FUNCTION_BLOCK StubXts EXTENDS Xts
VAR
END_VAR

METHOD Cycle : HRESULT
END_METHOD

METHOD Initialise : HRESULT
END_METHOD

METHOD MoverHomeSequence : BOOL
END_METHOD

METHOD SetDisabled : BOOL
VAR_INPUT
END_VAR
_XtsEnabled := FALSE;
END_METHOD

METHOD setEnabled : BOOL
VAR_INPUT
END_VAR
_XtsEnabled := TRUE;
END_METHOD

METHOD setInitialised : BOOL
VAR_INPUT
END_VAR
_Initialised := TRUE;
END_METHOD

METHOD setMoverNumberMax : BOOL
VAR_INPUT
END_VAR
_registeredNumberOfMovers := 255;
END_METHOD

METHOD setMoverNumberZero : BOOL
VAR_INPUT
END_VAR
_registeredNumberOfMovers := 0;
END_METHOD

METHOD setNotInitialised : BOOL
VAR_INPUT
END_VAR
_Initialised := FALSE;
END_METHOD

END_FUNCTION_BLOCK

(* stored: Version 1.1.0.1
   POU StubXts: Id {59a8f0f1-3a37-4f6e-9e76-a82474ad05c1}, SpecialFunc None
   Method Cycle: Id {ba7fc6ec-53fe-46e8-b7e8-7d8528b5c436}
   Method Initialise: Id {abac4287-77d3-4784-8f98-5b30950ef3e3}
   Method MoverHomeSequence: Id {75f313ff-91f0-4398-b273-e26bade55a8b}
   Method SetDisabled: Id {ffa0c583-2569-4ebd-98eb-9a7b4dc88c53}
   Method setEnabled: Id {626722de-9774-4f59-8220-0e027083d3f9}
   Method setInitialised: Id {2528f3aa-d996-4ef3-863b-9b23baf28b1f}
   Method setMoverNumberMax: Id {5d9d367e-74e6-410a-9121-5a46c3dda01c}
   Method setMoverNumberZero: Id {8cc461ce-7c43-4e66-86ca-dfa650521876}
   Method setNotInitialised: Id {fabc083b-0f7d-43b1-ade2-afd02e1ebe1b} *)
